PROGRAM P020_RtcEffectivityOEE
VAR
	//Wizka
	udiTotalCounter										:	UDINT;
	udiTotalefficiency									:	UDINT;

	//Rtc
	fbGetTime											:	NT_GetTime;				//FB getter RTC value
	tonDelay											:	TON;					//TON for delay between FB reading
	iCaseRtc											:	INT;					//Rtc case variable
	stActualTime										:	TIMESTRUCT;	

	wsActualDt											:	WSTRING := "00.00.0000 00:00:00";			
END_VAR

ACT_GetRtc();

ACTION ACT_GetRtc:
fbGetTime();
tonDelay(IN:=(iCaseRtc=2),PT:=T#200MS);
CASE iCaseRtc OF
	0:	//Start FB
		fbGetTime.START									:=	TRUE;
		iCaseRtc										:=	1;
	1:	//Wait #bysy signal
		IF (NOT fbGetTime.BUSY) THEN
			stActualTime								:=	fbGetTime.TIMESTR;
			fbGetTime.START								:=	FALSE;
			iCaseRtc									:=	2;
		END_IF
	2:	//Delay beetween reading RTC (for saving CPU time :) )
		IF (tonDelay.Q) THEN
			iCaseRtc									:=	0;
			wsActualDt:=METH_DateTimeArray_To_Wstring();
		END_IF
END_CASE
END_ACTION

METHOD METH_DateTimeArray_To_Wstring : WSTRING
VAR_INPUT
END_VAR
VAR 
	wsTmp												:	WSTRING;
END_VAR
IF (stActualTime.wDay<10) THEN
	wsTmp:="0";
END_IF
wsTmp:=WCONCAT(wsTmp,WCONCAT(UINT_TO_WSTRING(stActualTime.wDay),"."));

IF (stActualTime.wMonth<10) THEN
	wsTmp:=WCONCAT(wsTmp,"0");
END_IF
wsTmp:=WCONCAT(wsTmp,WCONCAT(UINT_TO_WSTRING(stActualTime.wMonth),"."));

IF (stActualTime.wYear<1000) THEN
	wsTmp:=WCONCAT(wsTmp,"0");
ELSIF (stActualTime.wYear<100) THEN
	wsTmp:=WCONCAT(wsTmp,"00");
ELSIF (stActualTime.wYear<10) THEN
	wsTmp:=WCONCAT(wsTmp,"000");
END_IF
wsTmp:=WCONCAT(wsTmp,WCONCAT(UINT_TO_WSTRING(stActualTime.wYear)," "));

IF (stActualTime.wHour<10) THEN
	wsTmp:=WCONCAT(wsTmp,"0");
END_IF
wsTmp:=WCONCAT(wsTmp,WCONCAT(UINT_TO_WSTRING(stActualTime.wHour),":"));
IF (stActualTime.wMinute<10) THEN
	wsTmp:=WCONCAT(wsTmp,"0");
END_IF
wsTmp:=WCONCAT(wsTmp,WCONCAT(UINT_TO_WSTRING(stActualTime.wMinute),":"));
IF (stActualTime.wSecond<10) THEN
	wsTmp:=WCONCAT(wsTmp,"0");
END_IF
wsTmp:=WCONCAT(wsTmp,UINT_TO_WSTRING(stActualTime.wSecond));
METH_DateTimeArray_To_Wstring:=wsTmp;
END_METHOD

END_PROGRAM

(* stored: Version 1.1.0.1, ProductVersion 3.1.4026.13, FileIdentifier c8fd074f6fa447948a269fdd1c2c5a7a71ef1b02, FileSignature 686a0a0fc4acefee64c5975f1665bf013b5581dd8cb7e39ba38f47c4d1e11c201aa5af6fc34db416b3c2e27ba1a725d94fd5f9742e122da6c9b953d9eaa81157e249b8422c6afc8a8988b18d718b7fb44bc5eac3a14ee0cf478b4ac9f62ab9e82601507634f2b557c7ade240d9e59f9a71a0dba353e65b513b0da78c8a9471cde69ae50ab4c35573f7b04faf38257946b63306ef653809a05228344d9ffa7f6f6d9b0379e829cb5e53320009be03ebea6d5a572bc9287c114c8e1e5f979df252a7d4bfa25c87f07add99faf499bd1029c66e2a87e40d493826a21e7c71ea7c7a5c793ce63fd47ce5f93d1c72d4c83f928fde59eccb642b57fcd395104d27a808
   POU P020_RtcEffectivityOEE: Id {c5d92e50-114d-4d8a-9269-718a2d11a074}, SpecialFunc None
   Action ACT_GetRtc: Id {b9b4b7cd-a07d-491d-b858-196ffa4e96fe}
   Method METH_DateTimeArray_To_Wstring: Id {611709b6-9d2b-43c1-80a8-cddb78c244c7} *)
